(* IEC 61131-3 sources: CodesysTest/alpha/export/PackML/OMAC/Function Blocks/UnitMode.pou/Commands, 10 files *)

(* ---- Abort.m.st ---- *)
(*#-#-#-#-#-#-#-#-#-#---Declaration---#-#-#-#-#-#-#-#-#-#-#-#-#*)

METHOD Abort : BOOL
VAR_INPUT
END_VAR
(*#-#-#-#-#-#-#-#-#-#---Implementation---#-#-#-#-#-#-#-#-#-#-#-#-#*)

CASE eState OF
PackMLState.Stopped,
PackMLState.Resetting,
PackMLState.Idle,
PackMLState.Starting,
PackMLState.Execute,
PackMLState.Holding,
PackMLState.Held,
PackMLState.UnHolding,
PackMLState.Suspending,
PackMLState.Suspended,
PackMLState.UnSuspending,
PackMLState.Completing,
PackMLState.Complete,
PackMLState.Stopping,
PackMLState.Clearing:
	IF (PackMLState.Aborting AND SupportedStates) = 0 THEN
		Abort := FALSE;
		RETURN;
	END_IF
	eState := PackMLState.Aborting;
	Abort := TRUE;
END_CASE

(* ---- ActingStateCompleted.m.st ---- *)
(*#-#-#-#-#-#-#-#-#-#---Declaration---#-#-#-#-#-#-#-#-#-#-#-#-#*)

// This method should be called by the program if an action has been finished.
METHOD ActingStateCompleted : BOOL
VAR_INPUT
END_VAR
(*#-#-#-#-#-#-#-#-#-#---Implementation---#-#-#-#-#-#-#-#-#-#-#-#-#*)

CASE eState OF
PackMLState.Holding,
PackMLState.UnHolding,
PackMLState.Starting,
PackMLState.Completing,
PackMLState.Resetting,
PackMLState.UnSuspending,
PackMLState.Suspending,
PackMLState.Aborting,
PackMLState.Stopping,
PackMLState.Clearing:
	IF (NextState(eState) AND SupportedStates) = 0 THEN
		ActingStateCompleted := FALSE;
		RETURN;
	END_IF
	eState := NextState(eState);
	ActingStateCompleted := TRUE;

PackMLState.Execute:
	IF (PackMLState.Completing AND SupportedStates) = 0 THEN
		ActingStateCompleted := FALSE;
		RETURN;
	END_IF
	eState := PackMLState.Completing;
	ActingStateCompleted := TRUE;
END_CASE

IF eState = PackMLState.Invalid THEN
	ActingStateCompleted := FALSE;
END_IF

(* ---- Clear.m.st ---- *)
(*#-#-#-#-#-#-#-#-#-#---Declaration---#-#-#-#-#-#-#-#-#-#-#-#-#*)

METHOD Clear : BOOL
VAR_INPUT
END_VAR
(*#-#-#-#-#-#-#-#-#-#---Implementation---#-#-#-#-#-#-#-#-#-#-#-#-#*)

CASE eState OF
PackMLState.Aborted:
	IF (PackMLState.Clearing AND SupportedStates) = 0 THEN
		Clear := FALSE;
		RETURN;
	END_IF
	eState := PackMLState.Clearing;
	Clear := TRUE;
END_CASE

(* ---- Hold.m.st ---- *)
(*#-#-#-#-#-#-#-#-#-#---Declaration---#-#-#-#-#-#-#-#-#-#-#-#-#*)

METHOD Hold : BOOL
VAR_INPUT
END_VAR
(*#-#-#-#-#-#-#-#-#-#---Implementation---#-#-#-#-#-#-#-#-#-#-#-#-#*)

CASE eState OF
PackMLState.Execute:
	IF (PackMLState.Holding AND SupportedStates) = 0 THEN
		Hold := FALSE;
		RETURN;
	END_IF
	eState := PackMLState.Holding;
	Hold := TRUE;
END_CASE

(* ---- Reset.m.st ---- *)
(*#-#-#-#-#-#-#-#-#-#---Declaration---#-#-#-#-#-#-#-#-#-#-#-#-#*)

METHOD Reset : BOOL
VAR_INPUT
END_VAR
(*#-#-#-#-#-#-#-#-#-#---Implementation---#-#-#-#-#-#-#-#-#-#-#-#-#*)

CASE eState OF
PackMLState.Complete,
PackMLState.Stopped:
	IF (PackMLState.Resetting AND SupportedStates) = 0 THEN
		Reset := FALSE;
		RETURN;
	END_IF
	eState := PackMLState.Resetting;
	Reset := TRUE;
END_CASE

(* ---- Start.m.st ---- *)
(*#-#-#-#-#-#-#-#-#-#---Declaration---#-#-#-#-#-#-#-#-#-#-#-#-#*)

METHOD Start : BOOL
VAR_INPUT
END_VAR
(*#-#-#-#-#-#-#-#-#-#---Implementation---#-#-#-#-#-#-#-#-#-#-#-#-#*)

CASE eState OF
PackMLState.Idle:
	IF (PackMLState.Starting AND SupportedStates) = 0 THEN
		Start := FALSE;
		RETURN;
	END_IF
	eState := PackMLState.Starting;
	Start := TRUE;
END_CASE

(* ---- Stop.m.st ---- *)
(*#-#-#-#-#-#-#-#-#-#---Declaration---#-#-#-#-#-#-#-#-#-#-#-#-#*)

METHOD Stop : BOOL
VAR_INPUT
END_VAR
(*#-#-#-#-#-#-#-#-#-#---Implementation---#-#-#-#-#-#-#-#-#-#-#-#-#*)

CASE eState OF
PackMLState.Resetting,
PackMLState.Idle,
PackMLState.Starting,
PackMLState.Execute,
PackMLState.Holding,
PackMLState.Held,
PackMLState.UnHolding,
PackMLState.Suspending,
PackMLState.Suspended,
PackMLState.UnSuspending,
PackMLState.Completing,
PackMLState.Complete:
	IF (PackMLState.Stopping AND SupportedStates) = 0 THEN
		Stop := FALSE;
		RETURN;
	END_IF
	eState := PackMLState.Stopping;
	Stop := TRUE;
END_CASE

(* ---- Suspend.m.st ---- *)
(*#-#-#-#-#-#-#-#-#-#---Declaration---#-#-#-#-#-#-#-#-#-#-#-#-#*)

METHOD Suspend : BOOL
VAR_INPUT
END_VAR
(*#-#-#-#-#-#-#-#-#-#---Implementation---#-#-#-#-#-#-#-#-#-#-#-#-#*)

CASE eState OF
PackMLState.Execute:
	IF (PackMLState.Suspending AND SupportedStates) = 0 THEN
		Suspend := FALSE;
		RETURN;
	END_IF
	eState := PackMLState.Suspending;
	Suspend := TRUE;
END_CASE

(* ---- UnHold.m.st ---- *)
(*#-#-#-#-#-#-#-#-#-#---Declaration---#-#-#-#-#-#-#-#-#-#-#-#-#*)

METHOD UnHold : BOOL
VAR_INPUT
END_VAR
(*#-#-#-#-#-#-#-#-#-#---Implementation---#-#-#-#-#-#-#-#-#-#-#-#-#*)

CASE eState OF
PackMLState.Held:
	IF (PackMLState.UnHolding AND SupportedStates) = 0 THEN
		UnHold := FALSE;
		RETURN;
	END_IF
	eState := PackMLState.UnHolding;
	UnHold := TRUE;
END_CASE

(* ---- UnSuspend.m.st ---- *)
(*#-#-#-#-#-#-#-#-#-#---Declaration---#-#-#-#-#-#-#-#-#-#-#-#-#*)

METHOD UnSuspend : BOOL
VAR_INPUT
END_VAR
(*#-#-#-#-#-#-#-#-#-#---Implementation---#-#-#-#-#-#-#-#-#-#-#-#-#*)

CASE eState OF
PackMLState.Suspended:
	IF (PackMLState.UnSuspending AND SupportedStates) = 0 THEN
		UnSuspend := FALSE;
		RETURN;
	END_IF
	eState := PackMLState.UnSuspending;
	UnSuspend := TRUE;
END_CASE
